(* CoDeSys 2.3.9.41 project: v0.10.pro *)
(* Libraries: STANDARD.LIB 5.6.98 12:03:02 *)

(* Task configuration *)
TASK Standard (PRIORITY := 0, INTERVAL := T#10ms);
	MAIN
END_TASK

(* Global variable list: Global_Variables *)
VAR_GLOBAL
	(*Digital Inputs*)
	bStart AT  %I* :BOOL;
	bStandby AT %I* :BOOL;
	bEmerency_Button AT %I*: BOOL;
	bEmergency_confirm AT %I*: BOOL;

	(*Digital outputs*)
	bStartLight AT  %Q* :BOOL;
	bStopLight AT %Q* :BOOL;
	bStandbyLight AT %Q* :BOOL;
	bEmergency_Light AT %Q*: BOOL;
	bStartup_power AT %Q*: BOOL;
	bBackup1 AT %Q* :BOOL;
	bBackup2 AT %Q* :BOOL;
	bBackup3 AT %Q* :BOOL;

	(*Analog inputs*)
	rAccelerationX AT %I* :INT;
	rAccelerationY AT %I* :INT;
	rAccelerationZ AT %I* :INT;
	rAnaloginputBackup AT %I* :INT;

	(*Analog Outputs*)
	iCylinderFL AT %Q* :INT;
	iCylinderFR AT %Q* :INT;
	iCylinderBLF AT %Q* :INT;
	iCylinderBLB AT %Q* :INT;
	iCylinderBRF AT %Q* :INT;
	iCylinderBRB AT %Q* :INT;
	iAnalogoutBackup1 AT %Q* :INT;
	iAnalogoutBackup2 AT %Q* :INT;

(*		Drawing of pneumatic cylinders in simulator
  
                                      FL/        \FR
		------------------------------------------
		|		Ambulace 		|
		|		Front			|
		|						|
		|						|
		|						|
		|						|
BLF	        /|						|\	BRF
	      /  |						|  \
	      \  |						|  /
	        \|						|/
BLB		|		rear				|	BRB
		|________________________|
		

*)
	(*Program variables*)


	FromADS:ARRAY [0..8] OF REAL;

	(*From Game*)
	LatAcc :REAL;
	LongAcc :REAL;
	HorizontalAcc:REAL;
	(*Not presently used*)
	Pitch:REAL;
	Roll:REAL;
	Speed:REAL;
	RPM:REAL;

	(*Testing for min-max values*)
	MaxX :REAL;
	MaxY:REAL;
	MaxZ:REAL;
	MinX :REAL;
	MinY:REAL;
	MinZ:REAL;


	(*Kirjota jotain fiksua*)
	rMultiplyerLatAcc:REAL;
	rMultiplyerLongAcc:REAL;
	rMultiplyerZAcc:REAL;
	rMultiplyerForce:REAL;
	rForceDirection:REAL;
	rCylinderFLCalc:REAL;
	rCylinderFRCalc:REAL;
	rCylinderBLFCalc:REAL;
	rCylinderBLBCalc:REAL;
	rCylinderBRFCalc:REAL;
	rCylinderBRBCalc:REAL;
	bEmergyStop_OK:BOOL;
	rpi: REAL;
	bEmergency_valvomo: BOOL;
	bStandby_Valvomo: BOOL;
	bStandby_internal: BOOL;
	bStart_Valvomo: BOOL;
	bStart_Internal: BOOL;
	bEmergency_Feedback: BOOL;
END_VAR

(* Global variable list: TwinCAT_Configuration *)
(* Generated automatically by TwinCAT - (read only) *)
VAR_CONFIG
	.bStart AT %IX8.0 : BOOL;
	.bStandby AT %IX8.1 : BOOL;
	.bEmerency_Button AT %IX8.2 : BOOL;
	.bEmergency_confirm AT %IX8.3 : BOOL;
	.bStartLight AT %QX16.0 : BOOL;
	.bStopLight AT %QX16.1 : BOOL;
	.bStandbyLight AT %QX16.2 : BOOL;
	.bEmergency_Light AT %QX16.3 : BOOL;
	.bStartup_power AT %QX16.4 : BOOL;
	.bBackup1 AT %QX16.5 : BOOL;
	.bBackup2 AT %QX16.6 : BOOL;
	.bBackup3 AT %QX16.7 : BOOL;
	.rAccelerationX AT %IB0 : INT;
	.rAccelerationY AT %IB2 : INT;
	.rAccelerationZ AT %IB4 : INT;
	.rAnaloginputBackup AT %IB6 : INT;
	.iCylinderFL AT %QB0 : INT;
	.iCylinderFR AT %QB2 : INT;
	.iCylinderBLF AT %QB4 : INT;
	.iCylinderBLB AT %QB6 : INT;
	.iCylinderBRF AT %QB8 : INT;
	.iCylinderBRB AT %QB10 : INT;
	.iAnalogoutBackup1 AT %QB12 : INT;
	.iAnalogoutBackup2 AT %QB14 : INT;
END_VAR

(* POU MAIN, FBD *)
PROGRAM MAIN
VAR
	M0: SR;
	M1: SR;
	M2: RS;
	M3: RS;

END_VAR
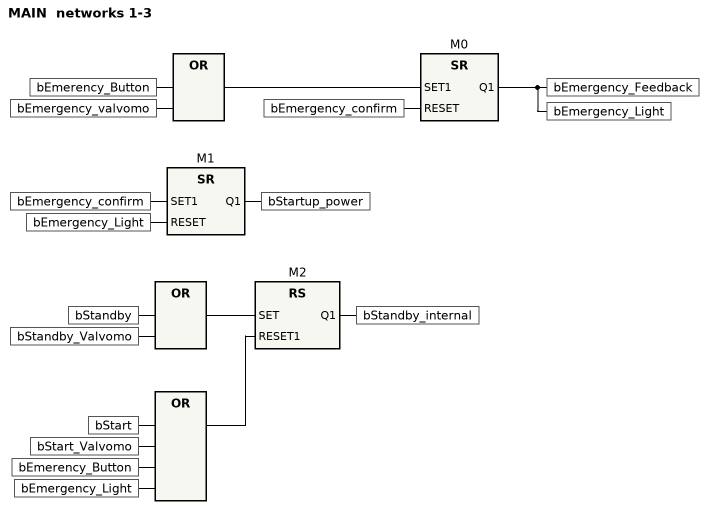
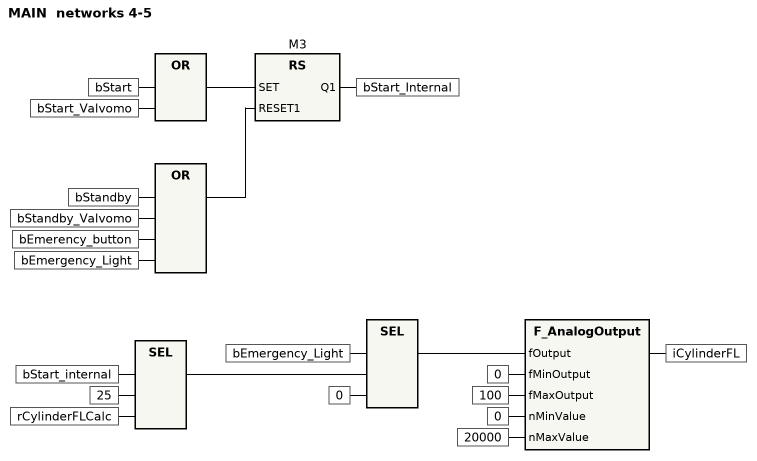
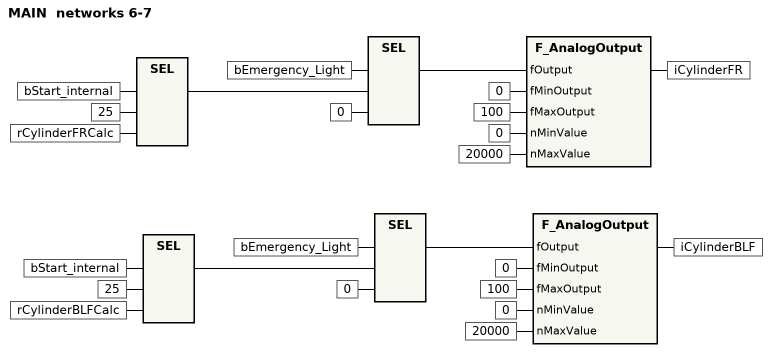
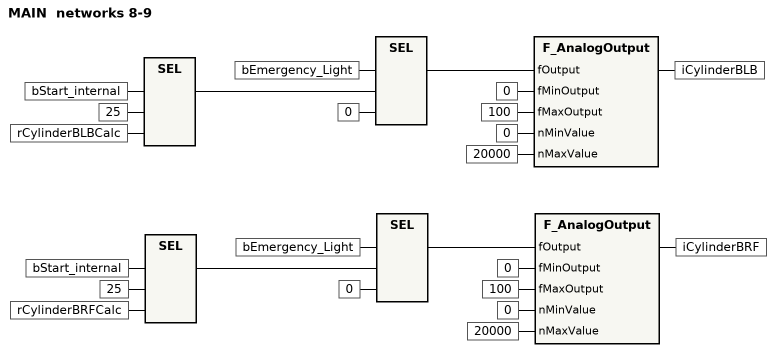
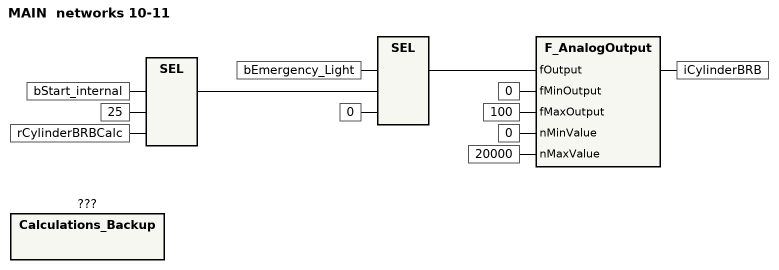
_FBD_ (* Function Block Diagram *)
NETWORK 1
	M0:SR(SET1: OR(bEmerency_Button, bEmergency_valvomo), RESET: bEmergency_confirm) => bEmergency_Feedback, bEmergency_Light
NETWORK 2
	M1:SR(SET1: bEmergency_confirm, RESET: bEmergency_Light) => bStartup_power
NETWORK 3
	M2:RS(SET: OR(bStandby, bStandby_Valvomo), RESET1: OR(bStart, bStart_Valvomo, bEmerency_Button, bEmergency_Light)) => bStandby_internal
NETWORK 4
	M3:RS(SET: OR(bStart, bStart_Valvomo), RESET1: OR(bStandby, bStandby_Valvomo, bEmerency_button, bEmergency_Light)) => bStart_Internal
NETWORK 5
	F_AnalogOutput(fOutput: SEL(bEmergency_Light, SEL(bStart_internal, 25, rCylinderFLCalc), 0), fMinOutput: 0, fMaxOutput: 100, nMinValue: 0, nMaxValue: 20000) => iCylinderFL
NETWORK 6
	F_AnalogOutput(fOutput: SEL(bEmergency_Light, SEL(bStart_internal, 25, rCylinderFRCalc), 0), fMinOutput: 0, fMaxOutput: 100, nMinValue: 0, nMaxValue: 20000) => iCylinderFR
NETWORK 7
	F_AnalogOutput(fOutput: SEL(bEmergency_Light, SEL(bStart_internal, 25, rCylinderBLFCalc), 0), fMinOutput: 0, fMaxOutput: 100, nMinValue: 0, nMaxValue: 20000) => iCylinderBLF
NETWORK 8
	F_AnalogOutput(fOutput: SEL(bEmergency_Light, SEL(bStart_internal, 25, rCylinderBLBCalc), 0), fMinOutput: 0, fMaxOutput: 100, nMinValue: 0, nMaxValue: 20000) => iCylinderBLB
NETWORK 9
	F_AnalogOutput(fOutput: SEL(bEmergency_Light, SEL(bStart_internal, 25, rCylinderBRFCalc), 0), fMinOutput: 0, fMaxOutput: 100, nMinValue: 0, nMaxValue: 20000) => iCylinderBRF
NETWORK 10
	F_AnalogOutput(fOutput: SEL(bEmergency_Light, SEL(bStart_internal, 25, rCylinderBRBCalc), 0), fMinOutput: 0, fMaxOutput: 100, nMinValue: 0, nMaxValue: 20000) => iCylinderBRB
NETWORK 11
	???:Calculations_Backup()
_END_FBD_
(* the same logic as Structured Text *)
(* Network 1 *)
M0(SET1 := bEmerency_Button OR bEmergency_valvomo, RESET := bEmergency_confirm);
bEmergency_Feedback := M0.Q1;
bEmergency_Light := M0.Q1;
(* Network 2 *)
M1(SET1 := bEmergency_confirm, RESET := bEmergency_Light);
bStartup_power := M1.Q1;
(* Network 3 *)
M2(SET := bStandby OR bStandby_Valvomo, RESET1 := bStart OR bStart_Valvomo OR bEmerency_Button OR bEmergency_Light);
bStandby_internal := M2.Q1;
(* Network 4 *)
M3(SET := bStart OR bStart_Valvomo, RESET1 := bStandby OR bStandby_Valvomo OR bEmerency_button OR bEmergency_Light);
bStart_Internal := M3.Q1;
(* Network 5 *)
iCylinderFL := F_AnalogOutput(fOutput := SEL(bEmergency_Light, SEL(bStart_internal, 25, rCylinderFLCalc), 0), fMinOutput := 0, fMaxOutput := 100, nMinValue := 0, nMaxValue := 20000);
(* Network 6 *)
iCylinderFR := F_AnalogOutput(fOutput := SEL(bEmergency_Light, SEL(bStart_internal, 25, rCylinderFRCalc), 0), fMinOutput := 0, fMaxOutput := 100, nMinValue := 0, nMaxValue := 20000);
(* Network 7 *)
iCylinderBLF := F_AnalogOutput(fOutput := SEL(bEmergency_Light, SEL(bStart_internal, 25, rCylinderBLFCalc), 0), fMinOutput := 0, fMaxOutput := 100, nMinValue := 0, nMaxValue := 20000);
(* Network 8 *)
iCylinderBLB := F_AnalogOutput(fOutput := SEL(bEmergency_Light, SEL(bStart_internal, 25, rCylinderBLBCalc), 0), fMinOutput := 0, fMaxOutput := 100, nMinValue := 0, nMaxValue := 20000);
(* Network 9 *)
iCylinderBRF := F_AnalogOutput(fOutput := SEL(bEmergency_Light, SEL(bStart_internal, 25, rCylinderBRFCalc), 0), fMinOutput := 0, fMaxOutput := 100, nMinValue := 0, nMaxValue := 20000);
(* Network 10 *)
iCylinderBRB := F_AnalogOutput(fOutput := SEL(bEmergency_Light, SEL(bStart_internal, 25, rCylinderBRBCalc), 0), fMinOutput := 0, fMaxOutput := 100, nMinValue := 0, nMaxValue := 20000);
(* Network 11: see the listing above *)
END_PROGRAM

(* POU Functions/F_AnalogOutput, ST *)
FUNCTION F_AnalogOutput : INT
VAR_INPUT
	fOutput: REAL; (* Output value *)
	fMinOutput:REAL; (* Scaling minimum value *)
	fMaxOutput:REAL; (* Scaling maximum value *)
	nMinValue: INT;  (* Maximum analog value *)
	nMaxValue: INT;  (* Maximum analog value *)
END_VAR
VAR
END_VAR
IF fOutput > fMaxOutput THEN
	fOutput := fMaxOutput;
ELSIF  fOutput < fMinOutput THEN
	fOutput := fMinOutput;
ELSIF  (fOutput >= fMinOutput) AND (fOutput <= fMaxOutput) THEN
	fOutput:= fOutput;
END_IF;

F_AnalogOutput := REAL_TO_INT((nMaxValue - nMinValue) * (fOutput - fMinOutput) / (fMaxOutput - fMinOutput) + nMinValue);
END_FUNCTION

(* POU Calculations_Backup, ST *)
PROGRAM Calculations_Backup
VAR
	P: BOOL;
END_VAR
rMultiplyerLongAcc:=2;
rMultiplyerLatAcc:=3;
rMultiplyerZAcc:=2;

LatAcc := FromADS[0];
HorizontalAcc := FromADS[1];
LongAcc := FromADS[2];

(*Testing with min-max values*)

MaxX := FromADS[3];
MaxY := FromADS[4];
MaxZ := FromADS[5];
MinX := FromADS[6];
MinY := FromADS[7];
MinZ := FromADS[8];

Pitch := 0;
Roll := 0;
Speed := 0;
RPM :=0;;
(* These are unused no, maybe will add them later
Pitch := FromADS[3];
Roll := FromADS[4];
Speed := FromADS[5];
RPM :=FromADS[6];
*)

rCylinderFLCalc:=LIMIT(0,rMultiplyerLongAcc*LongAcc-rMultiplyerLatAcc*LatAcc+rMultiplyerZAcc*HorizontalAcc+50,100);
rCylinderFRCalc:=LIMIT(0,rMultiplyerLongAcc*LongAcc+rMultiplyerLatAcc*LatAcc+rMultiplyerZAcc*HorizontalAcc+50,100);
rCylinderBLFCalc:=LIMIT(0,rMultiplyerZAcc*HorizontalAcc-rMultiplyerLongAcc*LongAcc*0.9-rMultiplyerLatAcc*LatAcc+50,100);
rCylinderBLBCalc:=LIMIT(0,rMultiplyerZAcc*HorizontalAcc-rMultiplyerLongAcc*LongAcc-rMultiplyerLatAcc*LatAcc+50,100);
rCylinderBRFCalc:=LIMIT(0,(rMultiplyerZAcc*HorizontalAcc-rMultiplyerLongAcc*LongAcc*0.9+rMultiplyerLatAcc*LatAcc+50),100);
rCylinderBRBCalc:=LIMIT(0,(rMultiplyerZAcc*HorizontalAcc-rMultiplyerLongAcc*LongAcc+rMultiplyerLatAcc*LatAcc+50),100);
END_PROGRAM

(* POU Calculations, ST *)
PROGRAM Calculations
VAR

	FLcalc: REAL;
	FRcalc:REAL;
	BLBcalc: REAL;
	BRBcalc: REAL;
	LongLat: REAL;
	apu1: REAL;
	apu2: REAL;
END_VAR
(*(*pi*)


(*Force calculations*)
IF LatAcc<>0 AND LongAcc<>0
THEN
MultiplyerForce:=SQRT(LatAcc*LatAcc+LongAcc*LongAcc);
END_IF;
(*direction calculations. First Exception*)
IF LatAcc=0
THEN
	IF  LongAcc>0
	THEN
	ForceDirection:=pi;
	ELSE
	ForceDirection:=0;
	END_IF;
ELSIF LongAcc=0
THEN
	IF  LatAcc>0
	THEN
	ForceDirection:=3/2*pi;
	ELSE
	ForceDirection:=pi/2;
	END_IF;
ELSE
LongLat:=LongAcc/LatAcc;
(*Direction calculations. Normal*)
	IF LongAcc>0 AND LatAcc>0
	THEN
	apu1:=ATAN(LongLat);
	apu2:=1.5*pi;
	ForceDirection:=apu2-apu1;

	ELSIF LongAcc<0 AND LatAcc>0
	THEN
	ForceDirection:=2*pi+ATAN(LongLat);

	ELSIF LongAcc<0 AND LatAcc<0
	THEN
	ForceDirection:=pi*0.5-ATAN(LongLat);

	ELSE
	ForceDirection:=pi+ATAN(LongLat);
	END_IF;
END_IF;
(*Cylinder output calculations*)
FLcalc:=ForceDirection;
FRcalc:=ForceDirection+(0.5*pi);
BLBcalc:=ForceDirection+(1.5*pi);
BRBcalc:=ForceDirection+pi;
CylinderFLCalc:=LIMIT(0,MultiplyerForce*SIN(FLcalc)+50+HorizontalAcc,100);
CylinderFRCalc:=LIMIT(0,MultiplyerForce*SIN(FRcalc)+50+HorizontalAcc,100);
(*CylinderBLFCalc:=LIMIT(0,MultiplyerForce*SIN(ForceDirection+2822)+50+HorizontalAcc,100);*)
CylinderBLBCalc:=LIMIT(0,MultiplyerForce*SIN(BLBcalc)+50+HorizontalAcc,100);
(*CylinderBRFCalc:=LIMIT(0,MultiplyerForce*SIN(ForceDirection+66566)+50+HorizontalAcc,100);*)
CylinderBRBCalc:=LIMIT(0,MultiplyerForce*SIN(BRBcalc)+50+HorizontalAcc,100);
(*nousee kääntäessä oikealle*)
*)


rpi:=3.141592654;
END_PROGRAM
